# B&R Automation Studio project mappPanel
Automation Studio 4.12.6.106; technology packages: mapp 5.24.3, mappView 5.24.4

## Configuration Sim

CPU PC_any, AutomationRuntime M4.93, Build 4.1.2, Safety 0.0, Vc V4.45.0

### Task classes (Cpu.sw)
```
Cyclic#4:
  TPanel <- mappPanel.TPanel.prg
DataObjects: BrowsePath <- mappPanel.BrowsePath.dob
Libraries: runtime, AsBrStr, sys_lib, standard, DataObj, AsOpcUac, AsOpcUas
```

### Hardware
```
PC : PC_any v1.1.1.0 (OrderNumber=PC)
  ConfigurationID = mappViewSample_Config1
  FileDevice1
  FileDeviceName1 = USER
  FileDevicePath1 = USER_PATH
  ActivateOpcUa = 1
  OpcUaInformationModels_PV_Version = 1
```

## Configuration X20CP

CPU X20CP3687X, AutomationRuntime M4.93, Build 4.1.2, Safety 0.0, Vc V4.45.0

### Task classes (Cpu.sw)
```
Cyclic#8:
  TPanel <- mappPanel.TPanel.prg
DataObjects: BrowsePath <- mappPanel.BrowsePath.dob
Binaries: mvLoader, udbdef, TCData, arconfig, User, Role, iomap, asfw, ashwac, ashwd, sysconf
Libraries: runtime, AsBrStr, sys_lib, standard, DataObj, AsOpcUac, AsOpcUas, astime, arssl, asieccon, fileio, IecCheck, AsICMP
```

### Hardware
```
6PPT80.156B-10A : 6PPT80.156B-10A v1.0.6.0  [ETH1 -> X20CP3687X.IF2 [Cable Type=PowerlinkCable, Length=10, Version=1.0.0.3]]
  Terminal = true
  PasswordVNC = 
  PasswordCIFS = 
  PasswordService = 
X20CP3687X : X20CP3687X v1.8.2.0
  Connector IF1:
    ActivateIna = 0
  Connector IF2:
    ActivateDevice = 1
    InaPort = 11160
    ActivateSnmp = 2
  ConfigurationID = mappViewSample_Config1
  FileDevice1
  FileDeviceName1 = USER
  FileDevicePath1 = USER_PATH
  ActivateSntpServer = 1
  ActivateOpcUa = 1
  OpcUaInformationModels_PV_Version = 1
```

## Logical view

Binary libraries used (declarations not repeated): operator, runtime, astime, AsIecCon, AsBrStr, sys_lib, standard, DataObj, AsOpcUac 6.5.0, AsOpcUas 6.5.0, IecCheck, AsICMP

### Package Logical/Libraries - Global libraries

- Visualisation Logical/mappView (not shown)

### Program Logical/mappPanel/TPanel (IEC)

#### TPanel.typ - Local data types
```iecst
TYPE
	StepEnum :
		(
		tpWAIT,
		tpCONNECT,
		tpDISCONNECT,
		tpPATH_GET,
		tpPATH_SAVE,
		tpSUBSCRIPTION,
		tpSUBSCRIPTION_DELETE,
		tpHANDLELIST,
		tpHANDLELIST_RELEASE,
		tpMONITORLIST,
		tpMONITORLIST_REMOVE,
		tpFIRST_READ,
		tpREADY,
		tpWRITE_TRANSLATE,
		tpWRITE_BULK,
		tpWRITE_WAIT,
		tpMETHOD_HANDLE,
		tpMETHOD_CALL,
		tpMETHOD_RELEASE,
		tpERROR,
		tpNONE
		);
	PowerPanelType : 	STRUCT
		Command : PowerPanelCmdType;
		Data : PowerPanelDataType;
		Parameter : PowerPanelParType;
		Method : MethodType;
		Diag : PowerPanelDiagType;
	END_STRUCT;
	PowerPanelCmdType : 	STRUCT
		Connect : BOOL;
		Disconnect : BOOL;
		Write : BOOL;
		ResetError : BOOL;
	END_STRUCT;
	PowerPanelDataType : 	STRUCT
		Startup : StartupType;
		Network : NetworkType;
		Time : TimeType;
		Screen : ScreenType;
		Audio : AudioType;
		Gesture : GestureType;
		Vnc : VncType;
		Web : WebType;
		Storage : StorageType;
		RemoteAccess : RemoteAccessType;
		AboutInfo : AboutInfoType;
		Diagnostics : DiagnosticsType;
		Status : StatusType;
		HandButton : GestureType;
	END_STRUCT;
	PowerPanelParType : 	STRUCT  (*Use one of the following types: T30, T50, FT50, T80*)
		PanelType : STRING[5];
		PanelIP : STRING[15];
	END_STRUCT;
	PowerPanelDiagType : 	STRUCT
		PingOk : BOOL;
		IsConnected : BOOL;
		PendingWrites : BOOL;
		Step : StepEnum;
		StatusText : STRING[200];
		StatusId : DWORD;
		VariableErrors : ARRAY[0..9]OF STRING[200];
		VariableErrorsIndex : USINT;
		VisHelperConnectVisible : BOOL;
		VisHelperErrorVisible : BOOL;
		ErrorStep : StepEnum := tpNONE;
	END_STRUCT;
	StartupType : 	STRUCT
		StartMode : UDINT;
		ShowBootLogoVNC : BOOL;
		ShowBootLogoWeb : BOOL;
		USBMemoryShare : BOOL;
		UserMemoryShare : BOOL;
	END_STRUCT;
	NetworkType : 	STRUCT
		Hostname : STRING[79];
		NetworkMode : UDINT;
		ActivateDNS : BOOL;
		DNSSuffix : STRING[79];
		GetDNSFromDHCP : BOOL;
		PrimaryDNS : STRING[79];
		SecondaryDNS : STRING[79];
		TertiaryDNS : STRING[79];
		IpAddress : STRING[79];
		SubnetMask : STRING[79];
		DefaultGateway : STRING[79];
	END_STRUCT;
	TimeType : 	STRUCT
		EnableNTPClient : BOOL;
		NTPServer1 : STRING[79];
		CurrentDateTime : DATE_AND_TIME;
	END_STRUCT;
	ScreenType : 	STRUCT
		DisplayBrightness : USINT;
		ScreenRotation : UDINT;
		EnableScreensaver : BOOL;
		ScreensaverIdleTime : UINT;
		ScreensaverType : UDINT;
	END_STRUCT;
	AudioType : 	STRUCT
		EnableBuzzer : BOOL;
		BuzzerSource : UDINT;
		BuzzerFrequency : UINT;
		BuzzerDuration : UINT;
	END_STRUCT;
	GestureType : 	STRUCT
		OpenServicePage : BOOL;
	END_STRUCT;
	DiagnosticsType : 	STRUCT
		CPUCore0Usage : USINT;
		CPUCore1Usage : USINT;
		CPUUsage : USINT;
		MemoryAvailable : UINT;
		MemoryTotal : UINT;
	END_STRUCT;
	VncType : 	STRUCT
		VNCServer : STRING[79];
		UseRfbExtension : BOOL;
		VNCLocalWindowScaling : BOOL;
		VNCBackgroundColor : STRING[79];
	END_STRUCT;
	WebType : 	STRUCT
		WebServer : STRING[79];
		VirtualKeyboardWeb : BOOL;
		DisablePinchGesture : BOOL;
		SetOverrideViewport : BOOL;
		ViewportSettings : STRING[79];
	END_STRUCT;
	StorageType : 	STRUCT
		USBMemoryShare : BOOL;
		UserMemoryShare : BOOL;
	END_STRUCT;
	RemoteAccessType : 	STRUCT
		EnableRemoteAccess : BOOL;
		RemoteAccessBackEnd : UDINT;
		RemoteAccessModeVNC : UDINT;
		RemoteAccessModeWebGL : UDINT;
		RemoteAccessPortWebGL : UINT;
		RemoteAccessWSPortWebGL : UINT;
		RemoteAccessPortVNC : UINT;
	END_STRUCT;
	AboutInfoType : 	STRUCT
		CompatibilityId : UDINT;
		DeviceRevision : STRING[79];
		HardwareRevision : STRING[79];
		Manufacturer : STRING[79];
		Model : STRING[79];
		ProductCode : UDINT;
		RevisionCounter : DINT;
		SerialNumber : STRING[79];
		SoftwareRevision : STRING[79];
		VendorId : UDINT;
	END_STRUCT;
	StatusType : 	STRUCT
		Temperature0 : REAL;
		Temperature1 : REAL;
		USBFlashDrive0 : UDINT;
		USBFlashDrive1 : UDINT;
	END_STRUCT;
	MethodType : 	STRUCT
		Type : PanelMethodType := NoMethod;
		BuzzerDuration : UDINT := 500;
		BuzzerFrequency : UDINT := 10000;
		ActualTime : STRING[79];
		Brightness : UDINT := 50;
	END_STRUCT;
	PanelMethodType :
		(
		NoMethod,
		AwakePanel,
		RestartSystem,
		StartRemoteAccess,
		StopRemoteAccess,
		SaveConfiguration,
		LoadConfiguration,
		StartUpdate,
		BuzzerDefault,
		BuzzerWithPara,
		SetBrightness,
		SetBrightnessUnlimited,
		SetTime
		);
	PvType : 	STRUCT
		ObjectIndex : INT;
		Adr : UDINT;
		AdrShadow : UDINT;
		DataLen : UDINT;
	END_STRUCT;
	BrowseType : 	STRUCT
		BrowsePath : STRING[79];
		VariableName : STRING[79];
		Argument : STRING[79];
		NamespaceIndex : UINT;
		Identifier : STRING[79];
		Access : STRING[1];
	END_STRUCT;
END_TYPE
```

#### TPanel.var - Local variables
```iecst
(*--------------------------------------------------------------------------------------------------------------------------------------------------------------------------------------------------------------------------------------------------------------------------------------------------------*)
(*Panel Configuration*)
(*--------------------------------------------------------------------------------------------------------------------------------------------------------------------------------------------------------------------------------------------------------------------------------------------------------*)
VAR RETAIN
	PanelIpAddress : STRING[15] := '192.168.30.180'; (*Panel IP address*)
	PanelType : STRING[15] := 'T80'; (*Use one of the following types: T30, T50, FT50, T80*)
END_VAR
(*--------------------------------------------------------------------------------------------------------------------------------------------------------------------------------------------------------------------------------------------------------------------------------------------------------*)
(*Error codes*)
(*--------------------------------------------------------------------------------------------------------------------------------------------------------------------------------------------------------------------------------------------------------------------------------------------------------*)
VAR CONSTANT
	ERR_PANEL_NO_DATA_MODULE : DWORD := 10000; (*The data module with the corresponding OPC UA tags is missing*)
	ERR_PANEL_IP_EMPTY : DWORD := 10001; (*IP address was not set*)
	ERR_PANEL_PANEL_TYPE_EMPTY : DWORD := 10002; (*Panel type was not set*)
	ERR_PANEL_FIRST_READ : DWORD := 10003; (*First read timed out*)
	ERR_PANEL_CONNECTION_LOST : DWORD := 10004; (*Connection to panel was interrupted*)
	ERR_PANEL_METHOD_NOT_FOUND : DWORD := 10005; (*The method does not exist on the corresponding panel*)
END_VAR
(*--------------------------------------------------------------------------------------------------------------------------------------------------------------------------------------------------------------------------------------------------------------------------------------------------------*)
(*Local constants*)
(*--------------------------------------------------------------------------------------------------------------------------------------------------------------------------------------------------------------------------------------------------------------------------------------------------------*)
VAR
	PING_TIMEOUT : UINT := 5000; (*Timeout for ping response*)
END_VAR
VAR CONSTANT
	INDEX_LIST : USINT := MAX_ELEMENTS_NODELIST-1;
END_VAR
(*--------------------------------------------------------------------------------------------------------------------------------------------------------------------------------------------------------------------------------------------------------------------------------------------------------*)
(*Local variables*)
(*--------------------------------------------------------------------------------------------------------------------------------------------------------------------------------------------------------------------------------------------------------------------------------------------------------*)
VAR
	Manufacturer : UALocalizedText;
	Model : UALocalizedText;
	PowerPanel : PowerPanelType;
	BrowseVar : {REDUND_UNREPLICABLE} BrowseType;
	pBrowseVar : REFERENCE TO BrowseType;
	TaskName : STRING[19];
	VariableStatus : UINT;
	VariableName : STRING[255];
	Device : STRING[79] := '';
	MethodSetBP : STRING[255];
	NodeErrorIdWrite : ARRAY[0..INDEX_LIST] OF DWORD := [MAX_ELEMENTS_NODELIST(0)];
	NodeQualityIDs : ARRAY[0..INDEX_LIST] OF DWORD;
	Offset : UDINT;
	MethodIndex : INT := 0;
	MethodPathLen : UINT;
	MethodCall : STRING[80] := '';
	PublishingInterval : TIME := T#3s;
	RemainingValueCount : ARRAY[0..INDEX_LIST] OF UINT;
	TimeStamps : ARRAY[0..INDEX_LIST] OF DATE_AND_TIME;
	ValuesChanged : ARRAY[0..INDEX_LIST] OF BOOL;
	VariablesReadInfo : ARRAY[0..INDEX_LIST] OF STRING[MAX_LENGTH_VARIABLE];
	VariablesTotalIndex : INT := 0;
	VariablesReadIndex : INT := 0;
	VariablesWriteIndex : INT := 0;
	VariablesChanged : ARRAY[0..INDEX_LIST] OF STRING[MAX_LENGTH_VARIABLE];
	VariablesChangeIndex : INT := 0;
	VariablesWriteInfo : ARRAY[0..INDEX_LIST] OF PvType;
	DataShadow : PowerPanelDataType;
	i : INT := 0;
	j : INT;
END_VAR
(*--------------------------------------------------------------------------------------------------------------------------------------------------------------------------------------------------------------------------------------------------------------------------------------------------------*)
(*Local function blocks*)
(*--------------------------------------------------------------------------------------------------------------------------------------------------------------------------------------------------------------------------------------------------------------------------------------------------------*)
VAR
	IcmpPing_0 : IcmpPing;
	PingTimer : TON_10ms;
	fbWaitAfterWrite : TON := (PT:=T#3s);
	fbFirstReadTimeout : TON_10ms := (PT:=1000);
	fbConnect : UA_Connect := (SessionConnectInfo:=(SessionName:='BuR',ApplicationName:='Panel',SecurityMsgMode:=UASecurityMsgMode_None,SecurityPolicy:=UASecurityPolicy_None,TransportProfile:=UATP_UATcp,UserIdentityToken:=(UserIdentityTokenType:=UAUITT_Anonymous),SessionTimeout:=T#1m,MonitorConnection:=T#30s));
	fbDisconnect : UA_Disconnect;
	fbMethodCall : UA_MethodCall;
	fbMethodGetHandle : UA_MethodGetHandle;
	fbMethodReleaseHandle : UA_MethodReleaseHandle;
	OutputArguments : ARRAY[0..9] OF UAMethodArgument;
	InputArguments : ARRAY[0..9] OF UAMethodArgument;
	fbTranslatePath : UA_TranslatePath;
	fbMonitoredItemAddList : UA_MonitoredItemAddList;
	fbMonitoredItemRemoveList : UA_MonitoredItemRemoveList;
	fbNodeGetHandleList : UA_NodeGetHandleList;
	fbNodeReleaseHandleList : UA_NodeReleaseHandleList;
	fbSubscriptionCreate : UA_SubscriptionCreate;
	fbSubscriptionDelete : UA_SubscriptionDelete;
	fbWriteBulk : UaClt_WriteBulk;
	MonitoringParameters : ARRAY[0..INDEX_LIST] OF UAMonitoringParameters;
	NodeAddInfoMonitor : ARRAY[0..INDEX_LIST] OF UANodeAdditionalInfo := [MAX_ELEMENTS_NODELIST((AttributeId:=UAAI_Value))];
	NodeAddInfoWrite : ARRAY[0..INDEX_LIST] OF UANodeAdditionalInfo := [MAX_ELEMENTS_NODELIST((AttributeId:=UAAI_Value))];
	UANodeIDMonitor : ARRAY[0..INDEX_LIST] OF UANodeID := [MAX_ELEMENTS_NODELIST(0)];
	UANodeIDWrite : ARRAY[0..INDEX_LIST] OF UANodeID := [MAX_ELEMENTS_NODELIST(0)];
	fbGetBrowsePath : DatObjInfo;
	fbWritePath : DatObjWrite := (enable:=TRUE);
END_VAR
```

#### Main.st - Cyclic code
```iecst
PROGRAM _CYCLIC
	// Make sure panel is reachable
	CheckPing;

	// Some helpers for the HMI
	PowerPanel.Diag.VisHelperConnectVisible := NOT PowerPanel.Diag.IsConnected;
	PowerPanel.Diag.VisHelperErrorVisible := PowerPanel.Diag.Step = tpERROR;

	// Some helpers for the OPC UA data
	PowerPanel.Data.AboutInfo.Manufacturer := Manufacturer.Text;
	PowerPanel.Data.AboutInfo.Model := Model.Text;

	// -----------------------------------------------------------------------------------------------------------------------------------------------------------------
	// Panel OPC UA connection state machine
	// -----------------------------------------------------------------------------------------------------------------------------------------------------------------
	CASE PowerPanel.Diag.Step OF

		// -----------------------------------------------------------------------------------------------------------------------------------------------------------------
		// IDLE state
		// -----------------------------------------------------------------------------------------------------------------------------------------------------------------
		tpWAIT:
			i := 0;
			PowerPanel.Diag.StatusText := 'Disconneted';
			PowerPanel.Diag.StatusId := 0;

			// -----------------------------------------------------------------------------------------------------------------------------------------------------------------
			// Wait for server to get ready
			IF (UaSrv_GetServerState() = UASS_Running) AND (PowerPanel.Diag.PingOk) AND (VariablesTotalIndex > 0) THEN

				// Wait for connect command
				IF PowerPanel.Command.Connect THEN
					// Make sure we have a valid IP address
					IF PowerPanel.Parameter.PanelIP = '' THEN
						PowerPanel.Diag.StatusId := ERR_PANEL_IP_EMPTY;
						PowerPanel.Diag.ErrorStep := PowerPanel.Diag.Step;
						PowerPanel.Diag.StatusText := 'IP address is empty';
						PowerPanel.Diag.Step := tpERROR;
						RETURN;
					END_IF

					// Make sure we have a valid panel type
					IF PowerPanel.Parameter.PanelType = '' THEN
						PowerPanel.Diag.StatusId := ERR_PANEL_PANEL_TYPE_EMPTY;
						PowerPanel.Diag.ErrorStep := PowerPanel.Diag.Step;
						PowerPanel.Diag.StatusText := 'Panel type is empty. Use one of the following types: T30, T50, FT50, T80';
						PowerPanel.Diag.Step := tpERROR;
						RETURN;
					END_IF

					brsmemset(ADR(UANodeIDMonitor), 0, SIZEOF(UANodeIDMonitor));
					brsmemset(ADR(fbTranslatePath), 0, SIZEOF(fbTranslatePath));
					brsmemset(ADR(fbSubscriptionCreate), 0, SIZEOF(fbSubscriptionCreate));
					brsmemset(ADR(fbMonitoredItemAddList), 0, SIZEOF(fbMonitoredItemAddList));
					brsmemset(ADR(fbNodeGetHandleList), 0, SIZEOF(fbNodeGetHandleList));
					brsmemset(ADR(PowerPanel.Diag.VariableErrors), 0, SIZEOF(PowerPanel.Diag.VariableErrors));
					PowerPanel.Diag.VariableErrorsIndex := 0;
					PowerPanel.Method.Type := NoMethod;

					// Prepare read variables
					brsmemset(ADR(MonitoringParameters), 0, SIZEOF(MonitoringParameters));
					FOR i := 0 TO INDEX_LIST DO
						MonitoringParameters[i].SamplingInterval := PublishingInterval;
						MonitoringParameters[i].Deadband := 0;
						MonitoringParameters[i].DeadbandType := UADeadbandType_None;
						MonitoringParameters[i].QueueSize := 0;
					END_FOR

					PowerPanel.Diag.StatusId := UINT_TO_DWORD(ERR_FUB_BUSY);
					PowerPanel.Diag.Step := tpCONNECT;
				END_IF
			END_IF

		// -----------------------------------------------------------------------------------------------------------------------------------------------------------------
		// Connect to panel via OPC
		// -----------------------------------------------------------------------------------------------------------------------------------------------------------------
		tpCONNECT:
			PowerPanel.Diag.StatusText := 'Connecting to panel...';

			// Set parameters for function call
			fbConnect.Execute := TRUE;
			fbConnect.ServerEndpointUrl := 'opc.tcp://';
			fbConnect.ServerEndpointUrl := CONCAT(fbConnect.ServerEndpointUrl, PowerPanel.Parameter.PanelIP);
			fbConnect.ServerEndpointUrl := CONCAT(fbConnect.ServerEndpointUrl, ':4840');
			fbConnect.Timeout := T#10s;

			// -----------------------------------------------------------------------------------------------------------------------------------------------------------------
			// Success
			IF fbConnect.Done THEN
				// Reset function block
				fbConnect.Execute := FALSE;

				// Set device and version string
				Device := '/0:Objects/2:DeviceSet/4:PowerPanel';
				Device := CONCAT(Device, PowerPanel.Parameter.PanelType);

				// Prepare path translation
				i := 0;
				Offset := 0;
				pBrowseVar ACCESS (fbGetBrowsePath.pDatObjMem + Offset);
				BrowseVar := pBrowseVar;
				brsmemset(ADR(fbTranslatePath.RelativePath), 0, SIZEOF(fbTranslatePath.RelativePath));

				PowerPanel.Diag.Step := tpPATH_GET;

			// -----------------------------------------------------------------------------------------------------------------------------------------------------------------
			// Go to error state
			ELSIF fbConnect.Error THEN
				fbConnect.Execute := FALSE;
				PowerPanel.Diag.StatusId := fbConnect.ErrorID;
				PowerPanel.Diag.StatusText := 'Error connecting to panel. ';
				IF PowerPanel.Diag.StatusId = 16#8005_0000 THEN
					brsstrcat(ADR(PowerPanel.Diag.StatusText), ADR('Make sure OPC UA server is activated.'));
				END_IF
				PowerPanel.Diag.ErrorStep := PowerPanel.Diag.Step;
				PowerPanel.Diag.Step := tpERROR;
			END_IF

			// -----------------------------------------------------------------------------------------------------------------------------------------------------------------
			// Function call

		// -----------------------------------------------------------------------------------------------------------------------------------------------------------------
		// Get path details
		// -----------------------------------------------------------------------------------------------------------------------------------------------------------------
		tpPATH_GET:
			PowerPanel.Diag.StatusText := 'Translating path...';

			// Set parameters for function call
			fbTranslatePath.Execute := TRUE;
			fbTranslatePath.ConnectionHdl := fbConnect.ConnectionHdl;
			fbTranslatePath.RelativePath := pBrowseVar.BrowsePath;
			fbTranslatePath.StartNodeID.Identifier := '84';
			fbTranslatePath.StartNodeID.IdentifierType := UAIdentifierType_Numeric;
			fbTranslatePath.Timeout := T#10s;

			IF (pBrowseVar.Access <> 'S') THEN
				fbTranslatePath.RelativePath := INSERT(fbTranslatePath.RelativePath, Device, 0);
			END_IF

			// -----------------------------------------------------------------------------------------------------------------------------------------------------------------
			// Success
			IF fbTranslatePath.Done THEN
				BrowseVar.NamespaceIndex := fbTranslatePath.TargetNodeID.NamespaceIndex;
				BrowseVar.Identifier := fbTranslatePath.TargetNodeID.Identifier;
				brsmemset(ADR(fbTranslatePath), 0, SIZEOF(fbTranslatePath));
				PowerPanel.Diag.Step := tpPATH_SAVE;

			// -----------------------------------------------------------------------------------------------------------------------------------------------------------------
			// Go to error state
			ELSIF fbTranslatePath.Error THEN
				fbTranslatePath.Execute := FALSE;
				// Variable is not available on this target
				IF (fbTranslatePath.ErrorID = 16#806F0000) OR (fbTranslatePath.ErrorID = 16#80AB0000) THEN
					PowerPanel.Diag.VariableErrors[PowerPanel.Diag.VariableErrorsIndex] := pBrowseVar.BrowsePath;
					IF PowerPanel.Diag.VariableErrorsIndex < SIZEOF(PowerPanel.Diag.VariableErrors)/SIZEOF(PowerPanel.Diag.VariableErrors[0]) - 1 THEN
						PowerPanel.Diag.VariableErrorsIndex := PowerPanel.Diag.VariableErrorsIndex + 1;
					END_IF
					PowerPanel.Diag.Step := tpPATH_SAVE;
				ELSE
					PowerPanel.Diag.StatusId := fbTranslatePath.ErrorID;
					PowerPanel.Diag.StatusText := 'Error translating path information';
					PowerPanel.Diag.ErrorStep := PowerPanel.Diag.Step;
					PowerPanel.Diag.Step := tpERROR;
				END_IF
			END_IF

		// -----------------------------------------------------------------------------------------------------------------------------------------------------------------
		// Save path information in data module
		// -----------------------------------------------------------------------------------------------------------------------------------------------------------------
		tpPATH_SAVE:
			PowerPanel.Diag.StatusText := 'Saving path...';

			// Set parameters for function call
			fbWritePath.enable := TRUE;
			fbWritePath.ident := fbGetBrowsePath.ident;
			fbWritePath.Offset := Offset;
			fbWritePath.pSource := ADR(BrowseVar);
			fbWritePath.len := SIZEOF(BrowseVar);
			fbWritePath();

			// -----------------------------------------------------------------------------------------------------------------------------------------------------------------
			// Success
			IF (fbWritePath.status = ERR_OK) THEN
				i := i + 1;

				// Translate path for next variable
				IF i < VariablesTotalIndex THEN
					Offset := i * SIZEOF(pBrowseVar);
					pBrowseVar ACCESS (fbGetBrowsePath.pDatObjMem + Offset);
					BrowseVar := pBrowseVar;
					brsmemset(ADR(fbTranslatePath.RelativePath), 0, SIZEOF(fbTranslatePath.RelativePath));
					PowerPanel.Diag.Step := tpPATH_GET;
				// Go to subscibe
				ELSE
					fbWritePath.enable := FALSE;

					DefineVariablesRead;
					DefineVariablesWrite;
					PowerPanel.Diag.Step := tpSUBSCRIPTION;
				END_IF

			// -----------------------------------------------------------------------------------------------------------------------------------------------------------------
			// Go to error state
			ELSIF (fbWritePath.status <> ERR_FUB_BUSY) THEN
				PowerPanel.Diag.StatusId := UINT_TO_DWORD(fbWritePath.status);
				PowerPanel.Diag.StatusText := 'Error saving path information';
				PowerPanel.Diag.ErrorStep := PowerPanel.Diag.Step;
				PowerPanel.Diag.Step := tpERROR;
			END_IF

		// -----------------------------------------------------------------------------------------------------------------------------------------------------------------
		// Start subsciption
		// -----------------------------------------------------------------------------------------------------------------------------------------------------------------
		tpSUBSCRIPTION:
			PowerPanel.Diag.StatusText := 'Subscribing...';

			// Set parameters for function call
			fbSubscriptionCreate.Execute := TRUE;
			fbSubscriptionCreate.ConnectionHdl := fbConnect.ConnectionHdl;
			fbSubscriptionCreate.Priority := 0;
			fbSubscriptionCreate.PublishingEnable := TRUE;
			fbSubscriptionCreate.Timeout := T#10s;

			// -----------------------------------------------------------------------------------------------------------------------------------------------------------------
			// Success
			IF fbSubscriptionCreate.Done THEN
				fbSubscriptionCreate.Execute := FALSE;
				PowerPanel.Diag.Step := tpHANDLELIST;

			// -----------------------------------------------------------------------------------------------------------------------------------------------------------------
			// Go to error state
			ELSIF fbSubscriptionCreate.Error THEN
				fbSubscriptionCreate.Execute := FALSE;
				PowerPanel.Diag.StatusId := fbSubscriptionCreate.ErrorID;
				PowerPanel.Diag.StatusText := 'Error subscribing to data';
				PowerPanel.Diag.ErrorStep := PowerPanel.Diag.Step;
				PowerPanel.Diag.Step := tpERROR;
			END_IF

		// -----------------------------------------------------------------------------------------------------------------------------------------------------------------
		// Get handles
		// -----------------------------------------------------------------------------------------------------------------------------------------------------------------
		tpHANDLELIST:
			PowerPanel.Diag.StatusText := 'Get handle list...';

			// Set parameters for function call
			fbNodeGetHandleList.Execute := TRUE;
			fbNodeGetHandleList.ConnectionHdl := fbConnect.ConnectionHdl;
			fbNodeGetHandleList.NodeIDs := UANodeIDMonitor;
			fbNodeGetHandleList.NodeIDCount := VariablesReadIndex;
			fbNodeGetHandleList.Timeout := T#10s;

			// -----------------------------------------------------------------------------------------------------------------------------------------------------------------
			// Success
			IF fbNodeGetHandleList.Done THEN
				fbNodeGetHandleList.Execute := FALSE;
				PowerPanel.Diag.Step := tpMONITORLIST;

				// -----------------------------------------------------------------------------------------------------------------------------------------------------------------
				// Go to error state
			ELSIF fbNodeGetHandleList.Error THEN
				fbNodeGetHandleList.Execute := FALSE;
				PowerPanel.Diag.StatusId := fbNodeGetHandleList.ErrorID;
				PowerPanel.Diag.StatusText := 'Error getting handle list. ';
				IF PowerPanel.Diag.StatusId = 16#800F_0000 THEN
					brsstrcat(ADR(PowerPanel.Diag.StatusText), ADR('Make sure panel type was set correct.'));
				END_IF

				// Find broken variable
				FOR i := 0 TO VariablesReadIndex DO
					IF fbMonitoredItemAddList.NodeErrorIDs[i] <> 0 THEN
						PowerPanel.Diag.StatusId := fbMonitoredItemAddList.NodeErrorIDs[i];
						PowerPanel.Diag.StatusText := VariablesReadInfo[i];
					END_IF
				END_FOR

				PowerPanel.Diag.ErrorStep := PowerPanel.Diag.Step;
				PowerPanel.Diag.Step := tpERROR;
			END_IF

		// -----------------------------------------------------------------------------------------------------------------------------------------------------------------
		// Start monitoring items
		// -----------------------------------------------------------------------------------------------------------------------------------------------------------------
		tpMONITORLIST:
			PowerPanel.Diag.StatusText := 'Start monitoring...';

			// Set parameters for function call
			fbMonitoredItemAddList.Execute := TRUE;
			fbMonitoredItemAddList.SubscriptionHdl := fbSubscriptionCreate.SubscriptionHdl;
			fbMonitoredItemAddList.NodeHdlCount := VariablesReadIndex;
			fbMonitoredItemAddList.NodeHdls := fbNodeGetHandleList.NodeHdls;
			fbMonitoredItemAddList.NodeAddInfos := NodeAddInfoMonitor;
			fbMonitoredItemAddList.Timeout := T#10s;

			// -----------------------------------------------------------------------------------------------------------------------------------------------------------------
			// Success
			IF fbMonitoredItemAddList.Done THEN
				fbMonitoredItemAddList.Execute := FALSE;

				// Reset first read timer
				fbFirstReadTimeout.IN := 0;
				fbFirstReadTimeout();

				PowerPanel.Diag.Step := tpFIRST_READ;

			// -----------------------------------------------------------------------------------------------------------------------------------------------------------------
			// Go to error state
			ELSIF fbMonitoredItemAddList.Error THEN
				fbMonitoredItemAddList.Execute := FALSE;
				PowerPanel.Diag.StatusId := fbMonitoredItemAddList.ErrorID;
				PowerPanel.Diag.StatusText := 'Error monitoring to data';

				// Find broken variable
				FOR i := 0 TO VariablesReadIndex DO
					IF fbMonitoredItemAddList.NodeErrorIDs[i] <> 0 THEN
						PowerPanel.Diag.StatusId := fbMonitoredItemAddList.NodeErrorIDs[i];
						PowerPanel.Diag.StatusText := VariablesReadInfo[i];
					END_IF
				END_FOR

				PowerPanel.Diag.ErrorStep := PowerPanel.Diag.Step;
				PowerPanel.Diag.Step := tpERROR;
			END_IF

		// -----------------------------------------------------------------------------------------------------------------------------------------------------------------
		// Wait for first data to arrive
		// -----------------------------------------------------------------------------------------------------------------------------------------------------------------
		tpFIRST_READ:
			PowerPanel.Diag.StatusText := 'Wait for first data...';

			fbFirstReadTimeout.IN := 1;
			fbFirstReadTimeout();

			// Panel did not respond with first data after 10s
			IF fbFirstReadTimeout.Q THEN
				PowerPanel.Diag.StatusId := ERR_PANEL_FIRST_READ;
				PowerPanel.Diag.ErrorStep := PowerPanel.Diag.Step;
				PowerPanel.Diag.StatusText := 'First read timed out';
				PowerPanel.Diag.Step := tpERROR;
			END_IF

			// Wait for first values to arrive
			IF PowerPanel.Data.AboutInfo.SerialNumber <> '' THEN
				// Create variable shadow for write variables
				FOR i := 0 TO VariablesWriteIndex - 1 DO
					brsmemcpy(VariablesWriteInfo[i].AdrShadow, VariablesWriteInfo[i].Adr, VariablesWriteInfo[i].DataLen);
				END_FOR

				PowerPanel.Diag.Step := tpREADY;
			END_IF

		// -----------------------------------------------------------------------------------------------------------------------------------------------------------------
		// Ready state with cyclic data exchange
		// -----------------------------------------------------------------------------------------------------------------------------------------------------------------
		tpREADY:
			// Set status and reset commands
			PowerPanel.Diag.StatusText := 'Ready';
			PowerPanel.Command.Connect := FALSE;
			PowerPanel.Command.ResetError := FALSE;
			PowerPanel.Diag.StatusId := 0;
			PowerPanel.Diag.IsConnected := TRUE;

			// -----------------------------------------------------------------------------------------------------------------------------------------------------------------
			// Track value changes
			CheckValueChange;
			IF VariablesChangeIndex > 0 AND PowerPanel.Command.Write THEN
				PowerPanel.Diag.StatusText := 'Writing new settings...';
				PowerPanel.Diag.Step := tpWRITE_BULK;
				RETURN;
			END_IF

			// -----------------------------------------------------------------------------------------------------------------------------------------------------------------
			// Method call handling
			IF PowerPanel.Method.Type <> NoMethod THEN
				PowerPanel.Diag.StatusText := 'Executing method...';
				DefineMethod;
				PowerPanel.Diag.StatusId := UINT_TO_DWORD(ERR_FUB_BUSY);
				PowerPanel.Diag.Step := tpMETHOD_HANDLE;
			END_IF

			// -----------------------------------------------------------------------------------------------------------------------------------------------------------------
			// Command disconnect
			IF PowerPanel.Command.Disconnect THEN
				PowerPanel.Diag.StatusText := 'Disconneting...';
				PowerPanel.Diag.StatusId := UINT_TO_DWORD(ERR_FUB_BUSY);
				PowerPanel.Diag.Step := tpMONITORLIST_REMOVE;
			END_IF

			// -----------------------------------------------------------------------------------------------------------------------------------------------------------------
			// Write all data that was changed
		// -----------------------------------------------------------------------------------------------------------------------------------------------------------------
		tpWRITE_BULK:
			// Set parameters for function call
			fbWriteBulk.Execute := TRUE;
			fbWriteBulk.ConnectionHdl := fbConnect.ConnectionHdl;
			fbWriteBulk.NodeIDCount := VariablesChangeIndex;
			fbWriteBulk.NodeIDs := ADR(UANodeIDWrite);
			fbWriteBulk.NodeAddInfo := ADR(NodeAddInfoWrite);
			fbWriteBulk.NodeErrorIDs := ADR(NodeErrorIdWrite);
			fbWriteBulk.Variables := ADR(VariablesChanged);

			// -----------------------------------------------------------------------------------------------------------------------------------------------------------------
			// Success
			IF fbWriteBulk.Done THEN
				fbWriteBulk.Execute := FALSE;
				PowerPanel.Diag.Step := tpWRITE_WAIT;

			// -----------------------------------------------------------------------------------------------------------------------------------------------------------------
			// Go to error state
			ELSIF fbWriteBulk.Error THEN
				fbWriteBulk.Execute := FALSE;
				PowerPanel.Diag.StatusId := fbWriteBulk.ErrorID;
				PowerPanel.Diag.StatusText := 'Error writing data';

				// Find broken variable
				FOR i := 0 TO VariablesChangeIndex DO
					IF NodeErrorIdWrite[i] <> 0 THEN
						PowerPanel.Diag.StatusId := NodeErrorIdWrite[i];
					END_IF
				END_FOR

				PowerPanel.Diag.ErrorStep := PowerPanel.Diag.Step;
				PowerPanel.Diag.Step := tpERROR;
			END_IF

		// -----------------------------------------------------------------------------------------------------------------------------------------------------------------
		// Wait for data to sink in
		// -----------------------------------------------------------------------------------------------------------------------------------------------------------------
		tpWRITE_WAIT:
			fbWaitAfterWrite.IN := TRUE;
			fbWaitAfterWrite();

			IF fbWaitAfterWrite.Q THEN
				fbWaitAfterWrite.IN := FALSE;
				fbWaitAfterWrite();

				// Create variable shadow for write variables
				FOR i := 0 TO VariablesWriteIndex - 1 DO
					brsmemcpy(VariablesWriteInfo[i].AdrShadow, VariablesWriteInfo[i].Adr, VariablesWriteInfo[i].DataLen);
				END_FOR

				// Reset command and flag
				PowerPanel.Command.Write := FALSE;
				PowerPanel.Diag.PendingWrites := FALSE;

				PowerPanel.Diag.Step := tpREADY;
			END_IF

		// -----------------------------------------------------------------------------------------------------------------------------------------------------------------
		// Get method handle
		// -----------------------------------------------------------------------------------------------------------------------------------------------------------------
		tpMETHOD_HANDLE:
			// Set parameters for function call
			fbMethodGetHandle.Execute := TRUE;
			fbMethodGetHandle.ConnectionHdl := fbConnect.ConnectionHdl;
			fbMethodGetHandle.Timeout := T#10s;

			// -----------------------------------------------------------------------------------------------------------------------------------------------------------------
			// Success
			IF fbMethodGetHandle.Done THEN
				fbMethodGetHandle.Execute := FALSE;
				PowerPanel.Diag.Step := tpMETHOD_CALL;

			// -----------------------------------------------------------------------------------------------------------------------------------------------------------------
			// Go to error state
			ELSIF fbMethodGetHandle.Error THEN
				fbMethodGetHandle.Execute := FALSE;
				PowerPanel.Diag.StatusId := fbMethodGetHandle.ErrorID;
				PowerPanel.Diag.StatusText := 'Error method handle';
				PowerPanel.Diag.ErrorStep := PowerPanel.Diag.Step;
				PowerPanel.Diag.Step := tpERROR;
			END_IF

		// -----------------------------------------------------------------------------------------------------------------------------------------------------------------
		// Call method
		// -----------------------------------------------------------------------------------------------------------------------------------------------------------------
		tpMETHOD_CALL:
			// Set parameters for function call
			fbMethodCall.Execute := TRUE;
			fbMethodCall.ConnectionHdl := fbConnect.ConnectionHdl;
			fbMethodCall.MethodHdl := fbMethodGetHandle.MethodHdl;
			fbMethodCall.Timeout := T#10s;

			// -----------------------------------------------------------------------------------------------------------------------------------------------------------------
			// Success
			IF fbMethodCall.Done THEN
				fbMethodCall.Execute := FALSE;
				PowerPanel.Diag.Step := tpMETHOD_RELEASE;

			// -----------------------------------------------------------------------------------------------------------------------------------------------------------------
			// Go to error state
			ELSIF fbMethodCall.Error THEN
				fbMethodCall.Execute := FALSE;
				PowerPanel.Diag.StatusId := fbMethodCall.ErrorID;
				PowerPanel.Diag.ErrorStep := PowerPanel.Diag.Step;
				PowerPanel.Diag.StatusText := 'Error executing method. Make sure parameter are correct';
				PowerPanel.Diag.Step := tpERROR;
			END_IF

		// -----------------------------------------------------------------------------------------------------------------------------------------------------------------
		// Release method handle
		// -----------------------------------------------------------------------------------------------------------------------------------------------------------------
		tpMETHOD_RELEASE:
			// Set parameters for function call
			fbMethodReleaseHandle.Execute := TRUE;
			fbMethodReleaseHandle.ConnectionHdl := fbConnect.ConnectionHdl;
			fbMethodReleaseHandle.MethodHdl := fbMethodGetHandle.MethodHdl;
			fbMethodReleaseHandle.Timeout := T#10s;

			// -----------------------------------------------------------------------------------------------------------------------------------------------------------------
			// Success
			IF fbMethodReleaseHandle.Done THEN
				fbMethodReleaseHandle.Execute := FALSE;

				// Disconnect when system was restarted
				IF PowerPanel.Method.Type = RestartSystem OR PowerPanel.Method.Type = StartUpdate THEN
					PowerPanel.Diag.Step := tpDISCONNECT;
				ELSE
					PowerPanel.Diag.Step := tpREADY;
				END_IF
				PowerPanel.Method.Type := NoMethod;

				// -----------------------------------------------------------------------------------------------------------------------------------------------------------------
			// Go to error state
			ELSIF fbMethodReleaseHandle.Error THEN
				fbMethodReleaseHandle.Execute := FALSE;
				PowerPanel.Diag.StatusId := fbMethodReleaseHandle.ErrorID;
				PowerPanel.Diag.StatusText := 'Error method release';
				PowerPanel.Diag.ErrorStep := PowerPanel.Diag.Step;
				PowerPanel.Diag.Step := tpERROR;
			END_IF

		// -----------------------------------------------------------------------------------------------------------------------------------------------------------------
		// Release monitored items
		// -----------------------------------------------------------------------------------------------------------------------------------------------------------------
		tpMONITORLIST_REMOVE:
			// Set parameters for function call
			fbMonitoredItemRemoveList.Execute := TRUE;
			fbMonitoredItemRemoveList.SubscriptionHdl := fbSubscriptionCreate.SubscriptionHdl;
			fbMonitoredItemRemoveList.MonitoredItemHdlCount := VariablesReadIndex;
			fbMonitoredItemRemoveList.MonitoredItemHdls := fbMonitoredItemAddList.MonitoredItemHdls;
			fbMonitoredItemRemoveList.Timeout := T#10s;

			// -----------------------------------------------------------------------------------------------------------------------------------------------------------------
			// Success
			IF fbMonitoredItemRemoveList.Done THEN
				fbMonitoredItemRemoveList.Execute := FALSE;
				PowerPanel.Diag.Step := tpSUBSCRIPTION_DELETE;

			// -----------------------------------------------------------------------------------------------------------------------------------------------------------------
			// Go to error state
			ELSIF fbMonitoredItemRemoveList.Error THEN
				fbMonitoredItemRemoveList.Execute := FALSE;
				PowerPanel.Diag.StatusId := fbMonitoredItemRemoveList.ErrorID;
				PowerPanel.Diag.StatusText := 'Error removing monitored items';
				PowerPanel.Diag.ErrorStep := PowerPanel.Diag.Step;
				PowerPanel.Diag.Step := tpERROR;
			END_IF

		// -----------------------------------------------------------------------------------------------------------------------------------------------------------------
		// Delet subsciption
		// -----------------------------------------------------------------------------------------------------------------------------------------------------------------
		tpSUBSCRIPTION_DELETE:
			// Set parameters for function call
			fbSubscriptionDelete.Execute := TRUE;
			fbSubscriptionDelete.SubscriptionHdl := fbSubscriptionCreate.SubscriptionHdl;
			fbSubscriptionDelete.Timeout := T#10s;

			// -----------------------------------------------------------------------------------------------------------------------------------------------------------------
			// Success
			IF fbSubscriptionDelete.Done THEN
				fbSubscriptionDelete.Execute := FALSE;
				PowerPanel.Diag.Step := tpHANDLELIST_RELEASE;

			// -----------------------------------------------------------------------------------------------------------------------------------------------------------------
			// Go to error state
			ELSIF fbSubscriptionDelete.Error THEN
				fbSubscriptionDelete.Execute := FALSE;
				PowerPanel.Diag.StatusId := fbSubscriptionDelete.ErrorID;
				PowerPanel.Diag.StatusText := 'Error deleting subscription';
				PowerPanel.Diag.ErrorStep := PowerPanel.Diag.Step;
				PowerPanel.Diag.Step := tpERROR;
			END_IF

		// -----------------------------------------------------------------------------------------------------------------------------------------------------------------
		// Release handles
		// -----------------------------------------------------------------------------------------------------------------------------------------------------------------
		tpHANDLELIST_RELEASE:
			// Set parameters for function call
			fbNodeReleaseHandleList.Execute := TRUE;
			fbNodeReleaseHandleList.ConnectionHdl := fbConnect.ConnectionHdl;
			fbNodeReleaseHandleList.NodeHdls := fbNodeGetHandleList.NodeHdls;
			fbNodeReleaseHandleList.NodeHdlCount := VariablesReadIndex;
			fbNodeReleaseHandleList.Timeout := T#10s;

			// -----------------------------------------------------------------------------------------------------------------------------------------------------------------
			// Success
			IF fbNodeReleaseHandleList.Done THEN
				fbNodeReleaseHandleList.Execute := FALSE;
				PowerPanel.Diag.Step := tpDISCONNECT;

			// -----------------------------------------------------------------------------------------------------------------------------------------------------------------
			// Go to error state
			ELSIF fbNodeReleaseHandleList.Error THEN
				fbNodeReleaseHandleList.Execute := FALSE;
				PowerPanel.Diag.StatusId := fbNodeReleaseHandleList.ErrorID;
				PowerPanel.Diag.StatusText := 'Error releasing handles';
				PowerPanel.Diag.ErrorStep := PowerPanel.Diag.Step;
				PowerPanel.Diag.Step := tpERROR;
			END_IF

		// -----------------------------------------------------------------------------------------------------------------------------------------------------------------
		// Disconnect from panel
		// -----------------------------------------------------------------------------------------------------------------------------------------------------------------
		tpDISCONNECT:
			// Set parameters for function call
			fbDisconnect.Execute := TRUE;
			fbDisconnect.ConnectionHdl := fbConnect.ConnectionHdl;
			fbDisconnect.Timeout := T#10s;

			// -----------------------------------------------------------------------------------------------------------------------------------------------------------------
			// Ignore errors during disconnect
			IF fbDisconnect.Done OR fbDisconnect.Error THEN
				fbDisconnect.Execute := FALSE;

				brsmemset(ADR(PowerPanel.Data), 0, SIZEOF(PowerPanel.Data));
				PowerPanel.Command.Disconnect := FALSE;
				PowerPanel.Diag.IsConnected := FALSE;
				fbDisconnect.Execute := FALSE;

				PowerPanel.Diag.Step := tpWAIT;
			END_IF

		// -----------------------------------------------------------------------------------------------------------------------------------------------------------------
		// Error state
		// -----------------------------------------------------------------------------------------------------------------------------------------------------------------
		tpERROR:
			PowerPanel.Command.Connect := FALSE;
			PowerPanel.Command.Disconnect := FALSE;

			// -----------------------------------------------------------------------------------------------------------------------------------------------------------------
			// Command error reset
			IF PowerPanel.Command.ResetError THEN
				PowerPanel.Diag.ErrorStep := tpNONE;
				PowerPanel.Diag.StatusId := 0;
				PowerPanel.Diag.StatusText := '';
				PowerPanel.Method.Type := NoMethod;
				PowerPanel.Command.ResetError := FALSE;

				IF PowerPanel.Diag.IsConnected THEN
					PowerPanel.Diag.Step := tpREADY;
				ELSE
					PowerPanel.Diag.Step := tpWAIT;
				END_IF
			END_IF
	END_CASE

	// -----------------------------------------------------------------------------------------------------------------------------------------------------------------
	// Function calls
	fbConnect();
	fbDisconnect();
	fbTranslatePath();
	fbSubscriptionCreate(PublishingInterval := PublishingInterval);
	fbNodeGetHandleList();
	fbMonitoredItemAddList(TimeStamps := TimeStamps, RemainingValueCount := RemainingValueCount, MonitoringSettings := MonitoringParameters, Variables := VariablesReadInfo, ValuesChanged := ValuesChanged, NodeQualityIDs := NodeQualityIDs);
	fbWriteBulk();
	fbMethodGetHandle();
	fbMethodCall(InputArguments := InputArguments, OutputArguments := OutputArguments);
	fbMethodReleaseHandle();
	fbMonitoredItemRemoveList();
	fbSubscriptionDelete();
	fbNodeReleaseHandleList();

END_PROGRAM
```

#### InitExit.st - Cyclic code
```iecst
PROGRAM _INIT
	// Transfer configuration
	PowerPanel.Parameter.PanelIP := PanelIpAddress;
	PowerPanel.Parameter.PanelType := PanelType;

	// Get task name
	ST_name(0,ADR(TaskName),0);
	PowerPanel.Data.Diagnostics.MemoryAvailable := 0;

	// Get data module details
	fbGetBrowsePath(enable := TRUE, pName := ADR('BrowsePath'));
	IF (fbGetBrowsePath.status = ERR_OK) THEN
		VariablesTotalIndex := UDINT_TO_INT(fbGetBrowsePath.len/SIZEOF(pBrowseVar));
	ELSE
		PowerPanel.Diag.StatusId := ERR_PANEL_NO_DATA_MODULE;
		PowerPanel.Diag.StatusText := 'no data module found';
		PowerPanel.Diag.Step := tpERROR;
	END_IF
END_PROGRAM

PROGRAM _EXIT
	REPEAT
		fbMonitoredItemRemoveList.Execute := TRUE;
		fbMonitoredItemRemoveList.SubscriptionHdl := fbSubscriptionCreate.SubscriptionHdl;
		fbMonitoredItemRemoveList.MonitoredItemHdlCount := VariablesReadIndex;
		fbMonitoredItemRemoveList.MonitoredItemHdls := fbMonitoredItemAddList.MonitoredItemHdls;
		fbMonitoredItemRemoveList();
		UNTIL NOT fbMonitoredItemRemoveList.Busy
	END_REPEAT
	REPEAT
		fbSubscriptionDelete.Execute := TRUE;
		fbSubscriptionDelete.SubscriptionHdl := fbSubscriptionCreate.SubscriptionHdl;
		fbSubscriptionDelete();
		UNTIL NOT fbSubscriptionDelete.Busy
	END_REPEAT
	REPEAT
		fbNodeReleaseHandleList.Execute := TRUE;
		fbNodeReleaseHandleList.ConnectionHdl := fbConnect.ConnectionHdl;
		fbNodeReleaseHandleList.NodeHdls := fbNodeGetHandleList.NodeHdls;
		fbNodeReleaseHandleList.NodeHdlCount := VariablesReadIndex;
		fbNodeReleaseHandleList();
		UNTIL NOT fbNodeReleaseHandleList.Busy
	END_REPEAT
	REPEAT
		fbDisconnect.Execute := TRUE;
		fbDisconnect.ConnectionHdl := fbConnect.ConnectionHdl;
		fbDisconnect();
		UNTIL NOT fbDisconnect.Busy
	END_REPEAT
END_PROGRAM
```

#### Action.st
```iecst
ACTION DefineVariablesRead:
	IF (fbGetBrowsePath.status = ERR_OK) THEN
		j := 0;
		FOR i := 0 TO VariablesTotalIndex - 1 DO
			pBrowseVar ACCESS (fbGetBrowsePath.pDatObjMem + (i * SIZEOF(pBrowseVar)));
			IF (pBrowseVar.Identifier <> '') AND (pBrowseVar.Access <> 'M') THEN
				UANodeIDMonitor[j].NamespaceIndex := pBrowseVar.NamespaceIndex;
				UANodeIDMonitor[j].IdentifierType := UAIdentifierType_Numeric;
				UANodeIDMonitor[j].Identifier := pBrowseVar.Identifier;
				VariablesReadInfo[j] := '::';
				VariablesReadInfo[j] := CONCAT(VariablesReadInfo[j], TaskName);
				VariablesReadInfo[j] := CONCAT(VariablesReadInfo[j], ':');
				VariablesReadInfo[j] := CONCAT(VariablesReadInfo[j], pBrowseVar.VariableName);
				j := j + 1;
			END_IF
			IF (j > INDEX_LIST) THEN
				EXIT;
			END_IF
		END_FOR
		IF j > 0 THEN
			VariablesReadIndex := j - 1;
		END_IF
	END_IF
END_ACTION

ACTION DefineVariablesWrite:
	DataShadow;
	IF (fbGetBrowsePath.status = ERR_OK) THEN
		j := 0;
		FOR i := 0 TO VariablesTotalIndex - 1 DO
			pBrowseVar ACCESS (fbGetBrowsePath.pDatObjMem + (i * SIZEOF(pBrowseVar)));
			IF (pBrowseVar.Identifier <> '') AND (pBrowseVar.Access = 'W') THEN
				// Get variable details
				VariablesWriteInfo[j].ObjectIndex := i;

				VariableName := '::';
				VariableName := CONCAT(VariableName, TaskName);
				VariableName := CONCAT(VariableName, ':');
				VariableName := CONCAT(VariableName, pBrowseVar.VariableName);
				VariableStatus := PV_xgetadr(ADR(VariableName), ADR(VariablesWriteInfo[j].Adr), ADR(VariablesWriteInfo[j].DataLen));

				// Make sure variable exists
				IF VariableStatus = 0 THEN
					VariableName := '::';
					VariableName := CONCAT(VariableName, TaskName);
					VariableName := CONCAT(VariableName, ':');
					VariableName := CONCAT(VariableName, REPLACE(pBrowseVar.VariableName, 'DataShadow', 15, 1));
					VariableStatus := PV_xgetadr(ADR(VariableName), ADR(VariablesWriteInfo[j].AdrShadow), ADR(VariablesWriteInfo[j].DataLen));

					j := j + 1;
				ELSE
					PowerPanel.Diag.StatusId := UINT_TO_DWORD(VariableStatus);
					PowerPanel.Diag.StatusText := VariableName;
					EXIT;
				END_IF

			END_IF
			IF (j > INDEX_LIST) THEN
				EXIT;
			END_IF
		END_FOR

		VariablesWriteIndex := j;
	END_IF
END_ACTION

ACTION CheckValueChange:
	PowerPanel.Diag.PendingWrites := FALSE;

	IF (fbGetBrowsePath.status = ERR_OK) THEN
		j := 0;
		brsmemset(ADR(VariablesChanged), 0 , SIZEOF(VariablesChanged));

		FOR i := 0 TO VariablesWriteIndex - 1 DO
			IF brsmemcmp(VariablesWriteInfo[i].Adr, VariablesWriteInfo[i].AdrShadow, VariablesWriteInfo[i].DataLen) <> 0 THEN
				pBrowseVar ACCESS (fbGetBrowsePath.pDatObjMem + (VariablesWriteInfo[i].ObjectIndex * SIZEOF(pBrowseVar)));
				UANodeIDWrite[j].Identifier := pBrowseVar.Identifier;
				UANodeIDWrite[j].NamespaceIndex := pBrowseVar.NamespaceIndex;
				UANodeIDWrite[j].IdentifierType := UAIdentifierType_Numeric;
				VariablesChanged[j] := VariablesReadInfo[VariablesWriteInfo[i].ObjectIndex];

				PowerPanel.Diag.PendingWrites := TRUE;

				j := j + 1;
				IF (j > INDEX_LIST) THEN
					EXIT;
				END_IF
			END_IF
		END_FOR

		VariablesChangeIndex := j;
	END_IF
END_ACTION

ACTION DefineMethod:
	// Set object ID
	FOR i:=0 TO VariablesTotalIndex - 1 DO
		pBrowseVar ACCESS (fbGetBrowsePath.pDatObjMem + (i * SIZEOF(pBrowseVar)));
		MethodIndex := FIND(pBrowseVar.BrowsePath,'/2:MethodSet');
		MethodPathLen := LEN(pBrowseVar.BrowsePath);
		IF (MethodIndex > 0) AND (MethodPathLen <= 12) THEN
			fbMethodGetHandle.ObjectNodeID.Identifier := pBrowseVar.Identifier;
			fbMethodGetHandle.ObjectNodeID.NamespaceIndex := pBrowseVar.NamespaceIndex;
			fbMethodGetHandle.ObjectNodeID.IdentifierType := UAIdentifierType_Numeric;
			EXIT;
		END_IF
	END_FOR
	MethodSetBP := '/2:MethodSet';

	// Set method ID parameters
	brsmemset(ADR(InputArguments),0,SIZEOF(InputArguments));
	IF PowerPanel.Method.Type = StartRemoteAccess THEN
		MethodCall := '/2:MethodSet/4:StartRemoteAccess';
	ELSIF PowerPanel.Method.Type = StopRemoteAccess THEN
		MethodCall := '/2:MethodSet/4:StopRemoteAccess';
	ELSIF PowerPanel.Method.Type = SaveConfiguration THEN
		MethodCall := '/2:MethodSet/4:SaveConfiguration';
	ELSIF PowerPanel.Method.Type = LoadConfiguration THEN
		MethodCall := '/2:MethodSet/4:LoadConfiguration';
	ELSIF PowerPanel.Method.Type = AwakePanel THEN
		MethodCall := '/2:MethodSet/4:AwakePanel';
	ELSIF PowerPanel.Method.Type = RestartSystem THEN
		MethodCall := '/2:MethodSet/4:RestartSystem';
	ELSIF PowerPanel.Method.Type = StartUpdate THEN
		MethodCall := '/2:MethodSet/4:StartUpdate';
	ELSIF PowerPanel.Method.Type = BuzzerDefault THEN
		MethodCall := '/2:MethodSet/4:BuzzerDefault';
	ELSIF PowerPanel.Method.Type = SetBrightness THEN
		MethodCall := '/2:MethodSet/4:SetBrightness';
	ELSIF PowerPanel.Method.Type = SetBrightnessUnlimited THEN
		MethodCall := '/2:MethodSet/4:SetBrightnessUnlimited';
	ELSIF PowerPanel.Method.Type = SetTime THEN
		MethodCall := '/2:MethodSet/4:SetTime';
	ELSIF PowerPanel.Method.Type = BuzzerWithPara THEN
		MethodCall := '/2:MethodSet/4:BuzzerWithPara';
	END_IF

	// Find method ID details
	FOR i:=0 TO (VariablesTotalIndex - 1) DO
		pBrowseVar ACCESS (fbGetBrowsePath.pDatObjMem + (i * SIZEOF(pBrowseVar)));
		MethodIndex := FIND(pBrowseVar.BrowsePath, MethodCall);
		IF (MethodIndex > 0) THEN
			fbMethodGetHandle.MethodNodeID.Identifier := pBrowseVar.Identifier;
			fbMethodGetHandle.MethodNodeID.NamespaceIndex := pBrowseVar.NamespaceIndex;
			fbMethodGetHandle.MethodNodeID.IdentifierType := UAIdentifierType_Numeric;

			IF PowerPanel.Method.Type = SetBrightness THEN
				MethodCall := '/2:MethodSet/4:SetBrightness';
				InputArguments[0].Name := 'Brightness';
				InputArguments[0].Value := '::';
				InputArguments[0].Value := CONCAT(InputArguments[0].Value,TaskName);
				InputArguments[0].Value := CONCAT(InputArguments[0].Value,':');
				InputArguments[0].Value := CONCAT(InputArguments[0].Value,pBrowseVar.VariableName);
			ELSIF PowerPanel.Method.Type = SetBrightnessUnlimited THEN
				MethodCall := '/2:MethodSet/4:SetBrightnessUnlimited';
				InputArguments[0].Name := 'BrightnessUnlimited';
				InputArguments[0].Value := '::';
				InputArguments[0].Value := CONCAT(InputArguments[0].Value,TaskName);
				InputArguments[0].Value := CONCAT(InputArguments[0].Value,':');
				InputArguments[0].Value := CONCAT(InputArguments[0].Value,pBrowseVar.VariableName);
			ELSIF PowerPanel.Method.Type = SetTime THEN
				MethodCall := '/2:MethodSet/4:SetTime';
				InputArguments[0].Name := 'Time';
				InputArguments[0].Value := '::';
				InputArguments[0].Value := CONCAT(InputArguments[0].Value,TaskName);
				InputArguments[0].Value := CONCAT(InputArguments[0].Value,':');
				InputArguments[0].Value := CONCAT(InputArguments[0].Value,pBrowseVar.VariableName);
			ELSIF PowerPanel.Method.Type = BuzzerWithPara THEN
				MethodCall := '/2:MethodSet/4:BuzzerWithPara';
				InputArguments[0].Name := 'Frequency';
				InputArguments[0].Value := '::';
				InputArguments[0].Value := CONCAT(InputArguments[0].Value,TaskName);
				InputArguments[0].Value := CONCAT(InputArguments[0].Value,':');
				InputArguments[0].Value := CONCAT(InputArguments[0].Value,pBrowseVar.VariableName);
				InputArguments[1].Name := 'Duration';
				InputArguments[1].Value := '::';
				InputArguments[1].Value := CONCAT(InputArguments[1].Value,TaskName);
				InputArguments[1].Value := CONCAT(InputArguments[1].Value,':');
				InputArguments[1].Value := CONCAT(InputArguments[1].Value,pBrowseVar.Argument);
			END_IF
			EXIT;
		END_IF
	END_FOR

	// Create error when method was not found
	IF MethodIndex = 0 THEN
		PowerPanel.Diag.StatusId := ERR_PANEL_METHOD_NOT_FOUND;
		PowerPanel.Diag.ErrorStep := PowerPanel.Diag.Step;
		PowerPanel.Diag.StatusText := 'Method type not found in data module';
		PowerPanel.Diag.Step := tpERROR;
	END_IF

END_ACTION

ACTION CheckPing:
	// Trigger ping request
	PingTimer.IN := TRUE;
	PingTimer.PT := PING_TIMEOUT;
	PingTimer();

	IcmpPing_0(enable := 1, pHost := ADR(PowerPanel.Parameter.PanelIP), timeout := PING_TIMEOUT);

	// Ping was OK
	IF(IcmpPing_0.status = ERR_OK) THEN
		PingTimer(IN := FALSE);
		PowerPanel.Diag.PingOk := TRUE;

	// Disconnect from share when ping failed
	ELSIF(IcmpPing_0.status <> ERR_FUB_BUSY) THEN
		PingTimer(IN := FALSE);
		PowerPanel.Diag.PingOk := FALSE;

		// Go to error state when connected
		IF PowerPanel.Diag.IsConnected THEN
			PowerPanel.Diag.IsConnected := FALSE;

			PowerPanel.Diag.StatusId := ERR_PANEL_CONNECTION_LOST;
			PowerPanel.Diag.ErrorStep := PowerPanel.Diag.Step;
			PowerPanel.Diag.StatusText := 'Connection is lost';
			PowerPanel.Diag.Step := tpERROR;
		END_IF
	END_IF
END_ACTION
```

### Data object Logical/mappPanel/BrowsePath (Simple)

#### BrowsePath.h
```c
#include <bur/plctypes.h>

typedef struct Browse_type
{
	plcstring BrowsePath[80];
	plcstring VariableName[80];
	plcstring Argument[80];
	unsigned short NamespaceIndex;
	plcstring Identifier[80];
	plcstring Access[2];
} BrowseType;
```

#### BrowsePath.c
```c
#include <BrowsePath.h>

struct Browse_type BrowseDat[] = {
	/*Browsepath,Variable/Argument,Argument,NameSpaceIndex,Identifier,Access*/
	{"/0:Objects/0:Server/0:ServerStatus/0:CurrentTime","PowerPanel.Data.Time.CurrentDateTime","",0x0000,"","S"},
	{"/3:Diagnostics/4:CPUCore0Usage","PowerPanel.Data.Diagnostics.CPUCore0Usage","",0x0000,"","R"},
	{"/3:Diagnostics/4:CPUCore1Usage","PowerPanel.Data.Diagnostics.CPUCore1Usage","",0x0000,"","R"},
	{"/3:Diagnostics/4:CPUUsage","PowerPanel.Data.Diagnostics.CPUUsage","",0x0000,"","R"},
	{"/3:Diagnostics/4:MemoryAvailable","PowerPanel.Data.Diagnostics.MemoryAvailable","",0x0000,"","R"},
	{"/3:Diagnostics/4:MemoryTotal","PowerPanel.Data.Diagnostics.MemoryTotal","",0x0000,"","R"},
	{"/3:Status/4:Temperature0","PowerPanel.Data.Status.Temperature0","",0x0000,"","R"},
	{"/3:Status/4:USBFlashDrive0","PowerPanel.Data.Status.USBFlashDrive0","",0x0000,"","R"},
	{"/3:Status/4:USBFlashDrive1","PowerPanel.Data.Status.USBFlashDrive1","",0x0000,"","R"},
	{"/2:Identification/3:CompatibilityId","PowerPanel.Data.AboutInfo.CompatibilityId","",0x0000,"","R"},
	{"/2:Identification/3:ProductCode","PowerPanel.Data.AboutInfo.ProductCode","",0x0000,"","R"},
	{"/2:Identification/3:VendorId","PowerPanel.Data.AboutInfo.VendorId","",0x0000,"","R"},
	{"/2:Identification/2:DeviceRevision","PowerPanel.Data.AboutInfo.DeviceRevision","",0x0000,"","R"},
	{"/2:Identification/2:HardwareRevision","PowerPanel.Data.AboutInfo.HardwareRevision","",0x0000,"","R"},
	{"/2:Identification/2:Manufacturer","Manufacturer","",0x0000,"","R"},
	{"/2:Identification/2:Model","Model","",0x0000,"","R"},
	{"/2:Identification/2:RevisionCounter","PowerPanel.Data.AboutInfo.RevisionCounter","",0x0000,"","R"},
	{"/2:Identification/2:SerialNumber","PowerPanel.Data.AboutInfo.SerialNumber","",0x0000,"","R"},
	{"/2:Identification/2:SoftwareRevision","PowerPanel.Data.AboutInfo.SoftwareRevision","",0x0000,"","R"},
	{"/3:Configuration/4:Startup/4:StartMode","PowerPanel.Data.Startup.StartMode","",0x0000,"","W"},
	{"/3:Configuration/4:Startup/4:ShowBootLogoVNC","PowerPanel.Data.Startup.ShowBootLogoVNC","",0x0000,"","W"},
	{"/3:Configuration/4:Startup/4:ShowBootLogoWeb","PowerPanel.Data.Startup.ShowBootLogoWeb","",0x0000,"","W"},
	{"/3:Configuration/4:Network/4:Hostname","PowerPanel.Data.Network.Hostname","",0x0000,"","W"},
	{"/3:Configuration/4:Network/4:NetworkMode","PowerPanel.Data.Network.NetworkMode","",0x0000,"","W"},
	{"/3:Configuration/4:Network/4:ActivateDNS","PowerPanel.Data.Network.ActivateDNS","",0x0000,"","W"},
	{"/3:Configuration/4:Network/4:DNSSuffix","PowerPanel.Data.Network.DNSSuffix","",0x0000,"","W"},
	{"/3:Configuration/4:Network/4:GetDNSFromDHCP","PowerPanel.Data.Network.GetDNSFromDHCP","",0x0000,"","W"},
	{"/3:Configuration/4:Network/4:PrimaryDNS","PowerPanel.Data.Network.PrimaryDNS","",0x0000,"","W"},
	{"/3:Configuration/4:Network/4:SecondaryDNS","PowerPanel.Data.Network.SecondaryDNS","",0x0000,"","W"},
	{"/3:Configuration/4:Network/4:TertiaryDNS","PowerPanel.Data.Network.TertiaryDNS","",0x0000,"","W"},
	{"/3:Configuration/4:Network/4:IpAddress","PowerPanel.Data.Network.IpAddress","",0x0000,"","W"},
	{"/3:Configuration/4:Network/4:SubnetMask","PowerPanel.Data.Network.SubnetMask","",0x0000,"","W"},
	{"/3:Configuration/4:Network/4:DefaultGateway","PowerPanel.Data.Network.DefaultGateway","",0x0000,"","W"},
	{"/3:Configuration/4:Time/4:EnableNTPClient","PowerPanel.Data.Time.EnableNTPClient","",0x0000,"","W"},
	{"/3:Configuration/4:Time/4:NTPServer1","PowerPanel.Data.Time.NTPServer1","",0x0000,"","W"},
	{"/3:Configuration/4:Screen/4:DisplayBrightness","PowerPanel.Data.Screen.DisplayBrightness","",0x0000,"","W"},
	{"/3:Configuration/4:Screen/4:ScreenRotation","PowerPanel.Data.Screen.ScreenRotation","",0x0000,"","W"},
	{"/3:Configuration/4:Screen/4:EnableScreensaver","PowerPanel.Data.Screen.EnableScreensaver","",0x0000,"","W"},
	{"/3:Configuration/4:Screen/4:ScreensaverIdleTime","PowerPanel.Data.Screen.ScreensaverIdleTime","",0x0000,"","W"},
	{"/3:Configuration/4:Screen/4:ScreensaverType","PowerPanel.Data.Screen.ScreensaverType","",0x0000,"","W"},
	{"/3:Configuration/4:Audio/4:EnableBuzzer","PowerPanel.Data.Audio.EnableBuzzer","",0x0000,"","W"},
	{"/3:Configuration/4:Audio/4:BuzzerSource","PowerPanel.Data.Audio.BuzzerSource","",0x0000,"","W"},
	{"/3:Configuration/4:Audio/4:BuzzerFrequency","PowerPanel.Data.Audio.BuzzerFrequency","",0x0000,"","W"},
	{"/3:Configuration/4:Audio/4:BuzzerDuration","PowerPanel.Data.Audio.BuzzerDuration","",0x0000,"","W"},
	{"/3:Configuration/4:Gesture/4:OpenServicePage","PowerPanel.Data.Gesture.OpenServicePage","",0x0000,"","W"},
	{"/3:Configuration/4:Vnc/4:VNCServer","PowerPanel.Data.Vnc.VNCServer","",0x0000,"","W"},
	{"/3:Configuration/4:Vnc/4:UseRfbExtension","PowerPanel.Data.Vnc.UseRfbExtension","",0x0000,"","W"},
	{"/3:Configuration/4:Vnc/4:VNCLocalWindowScaling","PowerPanel.Data.Vnc.VNCLocalWindowScaling","",0x0000,"","W"},
	{"/3:Configuration/4:Vnc/4:VNCBackgroundColor","PowerPanel.Data.Vnc.VNCBackgroundColor","",0x0000,"","W"},
	{"/3:Configuration/4:Web/4:WebServer","PowerPanel.Data.Web.WebServer","",0x0000,"","W"},
	{"/3:Configuration/4:Web/4:VirtualKeyboardWeb","PowerPanel.Data.Web.VirtualKeyboardWeb","",0x0000,"","W"},
	{"/3:Configuration/4:Web/4:SetOverrideViewport","PowerPanel.Data.Web.SetOverrideViewport","",0x0000,"","W"},
	{"/3:Configuration/4:Web/4:ViewportSettings","PowerPanel.Data.Web.ViewportSettings","",0x0000,"","W"},
	{"/3:Configuration/4:Web/4:DisablePinchGesture","PowerPanel.Data.Web.DisablePinchGesture","",0x0000,"","W"},
	{"/3:Configuration/4:Storage/4:USBMemoryShare","PowerPanel.Data.Storage.USBMemoryShare","",0x0000,"","W"},
	{"/3:Configuration/4:Storage/4:UserMemoryShare","PowerPanel.Data.Storage.UserMemoryShare","",0x0000,"","W"},
	{"/3:Configuration/4:RemoteAccess/4:EnableRemoteAccess","PowerPanel.Data.RemoteAccess.EnableRemoteAccess","",0x0000,"","W"},
	{"/3:Configuration/4:RemoteAccess/4:RemoteAccessBackEnd","PowerPanel.Data.RemoteAccess.RemoteAccessBackEnd","",0x0000,"","W"},
	{"/3:Configuration/4:RemoteAccess/4:RemoteAccessModeWebGL","PowerPanel.Data.RemoteAccess.RemoteAccessModeWebGL","",0x0000,"","W"},			// Requires firmware 1.6.0 or higher
	{"/3:Configuration/4:RemoteAccess/4:RemoteAccessModeVNC","PowerPanel.Data.RemoteAccess.RemoteAccessModeVNC","",0x0000,"","W"},				// Requires firmware 1.6.0 or higher
	{"/3:Configuration/4:RemoteAccess/4:RemoteAccessPortWebGL","PowerPanel.Data.RemoteAccess.RemoteAccessPortWebGL","",0x0000,"","W"},			// Requires firmware 1.6.0 or higher
	{"/3:Configuration/4:RemoteAccess/4:RemoteAccessWSPortWebGL","PowerPanel.Data.RemoteAccess.RemoteAccessWSPortWebGL","",0x0000,"","W"},		// Requires firmware 1.6.0 or higher
	{"/3:Configuration/4:RemoteAccess/4:RemoteAccessPortVNC","PowerPanel.Data.RemoteAccess.RemoteAccessPortVNC","",0x0000,"","W"},				// Requires firmware 1.6.0 or higher
	{"/2:MethodSet","","",0x0000,"","M"},
	{"/2:MethodSet/4:StartRemoteAccess","","",0x0000,"","M"},
	{"/2:MethodSet/4:StopRemoteAccess","","",0x0000,"","M"},
	{"/2:MethodSet/4:SaveConfiguration","","",0x0000,"","M"},
	{"/2:MethodSet/4:LoadConfiguration","","",0x0000,"","M"},
	{"/2:MethodSet/4:AwakePanel","","",0x0000,"","M"},
	{"/2:MethodSet/4:RestartSystem","","",0x0000,"","M"},																							// Requires firmware 1..0 or higher
	{"/2:MethodSet/4:StartUpdate","","",0x0000,"","M"},
	{"/2:MethodSet/4:BuzzerDefault","","",0x0000,"","M"},
	{"/2:MethodSet/4:SetBrightness","PowerPanel.Method.Brightness","",0x0000,"","M"},
	{"/2:MethodSet/4:SetBrightnessUnlimited","PowerPanel.Method.Brightness","",0x0000,"","M"},
	{"/2:MethodSet/4:SetTime","PowerPanel.Method.ActualTime","",0x0000,"","M"},
	{"/2:MethodSet/4:BuzzerWithPara","PowerPanel.Method.BuzzerFrequency","PowerPanel.Method.BuzzerDuration",0x0000,"","M"},
};
```

### revision.txt
```
28.11.2024
First release
```

### mappPanel.typ - not listed in the package file held
```iecst
TYPE
	mappPanelStepEnum :
		(
		tpWAIT,
		tpCONNECT,
		tpDISCONNECT,
		tpPATH_GET,
		tpPATH_SAVE,
		tpSUBSCRIPTION,
		tpSUBSCRIPTION_DELETE,
		tpHANDLELIST,
		tpHANDLELIST_RELEASE,
		tpMONITORLIST,
		tpMONITORLIST_REMOVE,
		tpFIRST_READ,
		tpREADY,
		tpWRITE_TRANSLATE,
		tpWRITE_BULK,
		tpWRITE_WAIT,
		tpMETHOD_HANDLE,
		tpMETHOD_CALL,
		tpMETHOD_RELEASE,
		tpERROR,
		tpNONE
		);
	PowerPanelType : 	STRUCT
		Command : PowerPanelCmdType;
		Data : PowerPanelDataType;
		Parameter : PowerPanelParType;
		Method : MethodType;
		Diag : PowerPanelDiagType;
	END_STRUCT;
	PowerPanelCmdType : 	STRUCT
		Connect : BOOL;
		Disconnect : BOOL;
		Write : BOOL;
		ResetError : BOOL;
	END_STRUCT;
	PowerPanelDataType : 	STRUCT
		Startup : StartupType;
		Network : NetworkType;
		Time : TimeType;
		Screen : ScreenType;
		Audio : AudioType;
		Gesture : GestureType;
		Vnc : VncType;
		Web : WebType;
		Storage : StorageType;
		RemoteAccess : RemoteAccessType;
		AboutInfo : AboutInfoType;
		Diagnostics : DiagnosticsType;
		Status : StatusType;
		HandButton : GestureType;
	END_STRUCT;
	PowerPanelParType : 	STRUCT  (*Use one of the following types: T30, T50, FT50, T80*)
		PanelType : STRING[5];
		PanelIP : STRING[15];
	END_STRUCT;
	PowerPanelDiagType : 	STRUCT
		PingOk : BOOL;
		IsConnected : BOOL;
		PendingWrites : BOOL;
		Step : mappPanelStepEnum;
		StatusText : STRING[200];
		StatusId : DWORD;
		VariableErrors : ARRAY[0..9]OF STRING[200];
		VariableErrorsIndex : USINT;
		VisHelperConnectVisible : BOOL;
		VisHelperErrorVisible : BOOL;
		ErrorStep : mappPanelStepEnum := (0);
	END_STRUCT;
	StartupType : 	STRUCT
		StartMode : UDINT;
		ShowBootLogoVNC : BOOL;
		ShowBootLogoWeb : BOOL;
		USBMemoryShare : BOOL;
		UserMemoryShare : BOOL;
	END_STRUCT;
	NetworkType : 	STRUCT
		Hostname : STRING[79];
		NetworkMode : UDINT;
		ActivateDNS : BOOL;
		DNSSuffix : STRING[79];
		GetDNSFromDHCP : BOOL;
		PrimaryDNS : STRING[79];
		SecondaryDNS : STRING[79];
		TertiaryDNS : STRING[79];
		IpAddress : STRING[79];
		SubnetMask : STRING[79];
		DefaultGateway : STRING[79];
	END_STRUCT;
	TimeType : 	STRUCT
		EnableNTPClient : BOOL;
		NTPServer1 : STRING[79];
		NTPServer2 : STRING[79];
		NTPServer3 : STRING[79];
		NTPServer4 : STRING[79];
		CurrentDateTime : DATE_AND_TIME;
	END_STRUCT;
	ScreenType : 	STRUCT
		DisplayBrightness : USINT;
		ScreenRotation : UDINT;
		EnableScreensaver : BOOL;
		ScreensaverIdleTime : UINT;
		ScreensaverType : UDINT;
		BootAnimationDelay : UINT;
		BootAnimationLeftPos : UINT;
		BootAnimationTopPos : UINT;
	END_STRUCT;
	AudioType : 	STRUCT
		EnableBuzzer : BOOL;
		BuzzerSource : UDINT;
		BuzzerFrequency : UINT;
		BuzzerDuration : UINT;
	END_STRUCT;
	GestureType : 	STRUCT
		OpenServicePage : BOOL;
		RestartSystem : BOOL;
	END_STRUCT;
	DiagnosticsType : 	STRUCT
		CPUCore0Usage : USINT;
		CPUCore1Usage : USINT;
		CPUUsage : USINT;
		MemoryAvailable : UINT;
		MemoryTotal : UINT;
	END_STRUCT;
	VncType : 	STRUCT
		VNCServer : STRING[79];
		UseRfbExtension : BOOL;
		VNCLocalWindowScaling : BOOL;
		VNCBackgroundColor : STRING[79];
		VNCConnectionMonitor : BOOL;
	END_STRUCT;
	WebType : 	STRUCT
		WebServer : STRING[79];
		VirtualKeyboardWeb : BOOL;
		DisablePinchGesture : BOOL;
		DisableGPU : BOOL;
		SetOverrideViewport : BOOL;
		ViewportSettings : STRING[79];
		IgnoreServerCertificateErrors : BOOL;
		EnableScreenCapture : BOOL;
		SuppressScrnCaptSecWarn : BOOL;
		WaitForNtpSync : BOOL;
		NtpSyncTimeout : UINT;
		SynchronizeTimeWithWebServer : BOOL;
	END_STRUCT;
	StorageType : 	STRUCT
		USBMemoryShare : BOOL;
		UserMemoryShare : BOOL;
	END_STRUCT;
	RemoteAccessType : 	STRUCT
		EnableRemoteAccess : BOOL;
		RemoteAccessBackEnd : UDINT;
		RemoteAccessModeVNC : UDINT;
		RemoteAccessModeWebGL : UDINT;
		RemoteAccessPortWebGL : UINT;
		RemoteAccessWSPortWebGL : UINT;
		RemoteAccessPortVNC : UINT;
	END_STRUCT;
	AboutInfoType : 	STRUCT
		CompatibilityId : UDINT;
		DeviceRevision : STRING[79];
		HardwareRevision : STRING[79];
		Manufacturer : STRING[79];
		Model : STRING[79];
		ProductCode : UDINT;
		SerialNumber : STRING[79];
		SoftwareRevision : STRING[79];
		VendorId : UDINT;
	END_STRUCT;
	StatusType : 	STRUCT
		Temperature0 : REAL;
		Temperature1 : REAL;
		USBFlashDrive0 : UDINT;
		USBFlashDrive1 : UDINT;
	END_STRUCT;
	MethodType : 	STRUCT
		Type : PanelMethodType := NoMethod;
		BuzzerDuration : UDINT := 500;
		BuzzerFrequency : UDINT := 10000;
		ActualTime : STRING[79];
		Brightness : UDINT := 50;
	END_STRUCT;
	PanelMethodType :
		(
		NoMethod,
		AwakePanel,
		RestartSystem,
		StartRemoteAccess,
		StopRemoteAccess,
		SaveConfiguration,
		LoadConfiguration,
		StartUpdate,
		BuzzerDefault,
		BuzzerWithPara,
		SetBrightness,
		SetBrightnessUnlimited,
		SetTime
		);
	PvType : 	STRUCT
		Name : STRING[MAX_LENGTH_VARIABLE];
		Writable : BOOL;
		ObjectIndex : INT;
		Adr : UDINT;
		AdrShadow : UDINT;
		DataLen : UDINT;
	END_STRUCT;
	BrowseType : 	STRUCT
		BrowsePath : STRING[79];
		VariableName : STRING[79];
		Argument : STRING[79];
		NamespaceIndex : UINT;
		Identifier : STRING[79];
		Access : STRING[1];
	END_STRUCT;
END_TYPE
```

### mappPanel.var - not listed in the package file held
```iecst
VAR
	PowerPanel : PowerPanelType;
END_VAR
(*--------------------------------------------------------------------------------------------------------------------------------------------------------------------------------------------------------------------------------------------------------------------------------------------------------*)
(*Panel Configuration*)
(*--------------------------------------------------------------------------------------------------------------------------------------------------------------------------------------------------------------------------------------------------------------------------------------------------------*)
VAR RETAIN
	PanelIpAddress : STRING[15] := '192.168.30.180'; (*Panel IP address*)
	PanelType : STRING[15] := 'T80'; (*Use one of the following types: T30, T50, FT50, T80*)
END_VAR
(*--------------------------------------------------------------------------------------------------------------------------------------------------------------------------------------------------------------------------------------------------------------------------------------------------------*)
(*Error codes*)
(*--------------------------------------------------------------------------------------------------------------------------------------------------------------------------------------------------------------------------------------------------------------------------------------------------------*)
VAR CONSTANT
	ERR_PANEL_NO_DATA_MODULE : DWORD := 10000; (*The data module with the corresponding OPC UA tags is missing*)
	ERR_PANEL_IP_EMPTY : DWORD := 10001; (*IP address was not set*)
	ERR_PANEL_PANEL_TYPE_EMPTY : DWORD := 10002; (*Panel type was not set*)
	ERR_PANEL_FIRST_READ : DWORD := 10003; (*First read timed out*)
	ERR_PANEL_CONNECTION_LOST : DWORD := 10004; (*Connection to panel was interrupted*)
	ERR_PANEL_METHOD_NOT_FOUND : DWORD := 10005; (*The method does not exist on the corresponding panel*)
	ERR_PANEL_INDEX_EXCEEDED : DWORD := 10006; (*Maximum number of variables subscription reached (64)*)
END_VAR
```

Listed in the project but not available here: Logical/Global.typ
